{attribute 'qualified_only'}
VAR_GLOBAL
	sNetId: T_AmsNetId := '5.53.143.17.1.1';
	nPort: T_AmsPort := 851;	
END_VAR

(* stored: Version 1.1.0.1, ProductVersion 3.1.4024.11
   GVL StripperAms: Id {f36a9f62-bf8a-4cb8-8c8c-493d69e2d7b9} *)
